// TwinCAT 3 PLC project ProviderPLC
// ProgramVersion: 3.1.4026.22
// libraries:
//   Tc2_EtherCAT, * (Beckhoff Automation GmbH)
//   Tc2_Standard, * (Beckhoff Automation GmbH)
//   Tc2_System, * (Beckhoff Automation GmbH)
//   Tc3_RealtimeMonitoring, * (Beckhoff Automation GmbH)
// project tree:
//   POUs/ FB_DoWork.TcPOU, F_ConsumeTime.TcPOU (not stored), MAIN.TcPOU
//   / ProviderPLC.TcTTO
// (motion and I/O tree: see PLC project plc1)
// real-time tasks:
//   TASK Plc1Task: cycle T#10ms, priority 20, ADS port 350
//   TASK Plc2Task: cycle T#10ms, priority 21, ADS port 351
//   TASK ProviderPLC: cycle T#10ms, priority 13, ADS port 352
// variable links:
//   (this object) <-> ProviderPLC/ProviderPLC Instance
//     PlcTask Inputs/MAIN.fbDoWorkProxy.nObjId <-> ProviderPLC Outputs/MAIN.fbDoWork.objID

CONFIGURATION ProviderPLC
    RESOURCE PLC ON TwinCAT3
        TASK ProviderPLC(INTERVAL := T#10ms, PRIORITY := 13);
        PROGRAM MAIN WITH ProviderPLC : MAIN;
    END_RESOURCE
END_CONFIGURATION

// ---- POUs/MAIN.TcPOU
//Provider PLC
PROGRAM MAIN
VAR
	DelayToCallInterface : UDINT := 10;
	fbDoWork			 : FB_DoWork('MAIN.fbDoWork');
END_VAR

F_ConsumeTime(DelayToCallInterface);
fbDoWork.M_Increment();

END_PROGRAM

// ---- POUs/FB_DoWork.TcPOU
{attribute 'c++_compatible'}
FUNCTION_BLOCK FB_DoWork EXTENDS TcBaseModuleRegistered IMPLEMENTS I_DoWork

METHOD FB_reinit : BOOL
SUPER^.FB_reinit();
END_METHOD

{attribute 'TcTypeSystem'}
{attribute 'c++_compatible'}
{attribute 'minimal_input_size' := '4'}
{attribute 'pack_mode' := '4'}
METHOD M_Increment : Global.HRESULT
VAR_INST
	fbCrititcalSection : FB_IecCriticalSection;
	fbRTMon_LogMark	   : FB_RTMon_LogMark;
	_counter		   : UDINT;	
END_VAR
IF fbCrititcalSection.Enter() THEN
	(* start of critical section *)
	fbRTMon_LogMark.LogStart(0, 0);
	_counter := _counter + 1;
	F_ConsumeTime(100);
	M_Increment := S_OK;
	fbRTMon_LogMark.LogStop(0, 0);

	(* end of critical section *)
	fbCrititcalSection.Leave();
END_IF
END_METHOD

{attribute 'minimal_input_size' := '4'}
{attribute 'pack_mode' := '4'}
{attribute 'c++_compatible'}
METHOD TcQueryInterface : Tc3_Module.HRESULT
VAR_INPUT
	iid	   : REFERENCE TO Tc3_Module.IID;
	pipItf : POINTER TO Tc3_Module.PVOID;
END_VAR

VAR
	ipDoWork : I_DoWork;
END_VAR
IF GuidsEqual(ADR(iid), ADR(TC_GLOBAL_IID_LIST.IID_I_DoWork)) THEN
	ipDoWork := THIS^; // cast to interface pointer
	pipItf^ := ITCUNKNOWN_TO_PVOID(ipDoWork);
	TcAddRef();
	TcQueryInterface := S_OK;
ELSE
	TcQueryInterface := SUPER^.TcQueryInterface(iid, pipItf);
END_IF
END_METHOD

END_FUNCTION_BLOCK
